PROGRAM MAIN
VAR{varable needed}
	robot				: FB_Robot;
	fbReadAxisStatus 	: FB_ReadAxisStatus;
	fbMCMotion 			: ARRAY[0..19] OF FB_SetAxisMotion;
	
	MC_ActStatus		: st_AxisGroupRead; 		 //**OUT**give the data to thr Upper
	MC_SetCommd			: st_AxisGroupSet;			 //**IN** get the data from the Upper and set the Axis 
	CtlComd		: RecvBuff;		(*Commd to MC*)
	Status		: SendBuff;		(*MC_State*)
	
	
	ErrID		: UDINT := 0;	
	step		: INT := 0;
	{time cost of every cycle}
	CycleTime	: LREAL := 0;
	CycleTime_Max: LREAL := 0;	
END_VAR

VAR{varable FOR test}
	i :UDINT := 0;
	j :UDINT := 0;
	w :UDINT := 0;
	vel : LREAL;
	nCounter: BYTE := 0;
	nCounter1: BYTE := 0;
	GetTime:GETCPUACCOUNT;
	time_start: UDINT;
	time_end:UDINT;
	labelOld:DINT := 0;
	labelNew:DINT := 0;
	count: UDINT := 0;
	count11 : UDINT := 0;
	delay : TON;
	
	test : LREAL := 0;
	test1 : LREAL := 0;
END_VAR

CASE step OF
	0: {prepare varable before start robot}	
		step := 5;
	5:	{NC init before robot start}	
		GroupInitAxis(); 	
		step := 10;
	10:{Init robot}
		ErrID := robot.InitRobot(ADR(GVL.InitPar));
	 	IF (0 = ErrID )THEN
		 	step := 15;
		ELSE
			step := 0;
		END_IF
	15:
		GetTime(cpuAccountDW=>time_start);
	 	
		GVL.fbRecvDataQue.GetfromQue(ADR(CtlComd));
		GroupReadAxis();

		robot.RunRobot(pMC_Inputs := ADR(MC_ActStatus), pMC_Outputs := ADR(MC_SetCommd),
								pCtlComd	:= ADR(CtlComd) , pRobotStatus := ADR(Status));
														
		GroupSetAxis();
		GVL.fbSendDataQue.PutToQue(ADR(Status));
		
		GetTime(cpuAccountDW=>time_end);
		CycleTime := (time_end- time_start)/10000.0;
		CycleTime_Max:= MAX(CycleTime,CycleTime_Max);
	 	
	20: 
		robot.StopRobot();
		step:= 0;
END_CASE;

ACTION GroupInitAxis:
i := 0;
END_ACTION

ACTION GroupReadAxis:
FOR i:= 0 TO 7 DO //MC_ActStatus.Number
	fbReadAxisStatus(AxisRef := GVL.TestMotor[i], AxisStatus => MC_ActStatus.AxisGoup[i]);	
END_FOR
END_ACTION

ACTION GroupSetAxis:
FOR i:= 0 TO 7 DO //MC_ActStatus.Number
	fbMCMotion[i](axis := GVL.TestMotor[i], SetCmd := MC_SetCommd.AxisGroup[i], ActStatus := MC_ActStatus.AxisGoup[i]);
END_FOR
//fbMCMotion(axis := GVL.TestMotor[0], SetCmd := MC_SetCommd.AxisGroup[0], ActStatus := MC_ActStatus.AxisGoup[0]);
END_ACTION

END_PROGRAM

(* stored: Version 1.1.0.1, ProductVersion 3.1.4022.12
   POU MAIN: Id {c3a5645a-c88b-4d8d-9c7f-23d853324ec7}, SpecialFunc None
   Action GroupInitAxis: Id {9457ddde-3e72-4440-a7d5-33bae3ae3ccf}
   Action GroupReadAxis: Id {14c0d48f-5ba2-4ac9-9f47-d99d60eeb3df}
   Action GroupSetAxis: Id {136d041d-cbc5-43ae-8121-b996fcb4942e} *)
